// TIA Portal V20 export
TYPE "Equipment"
   STRUCT
      "type" : Int;
      commandOn : Bool;
      commandOff : Bool;
      feedbackOn : Bool;
      feedbackOff : Bool;
      isFaulty : Bool;
      isProcessFinished : Bool;
   END_STRUCT;
END_TYPE
